// TIA Portal V20 export
TYPE "LKinCtrl_typeAdvPointers"
   STRUCT
      addPointer : DInt := 0;   // pointer to add new comds to PathData after cmd has been executed by MovePath
      retrievePointer : DInt := 0;   // pointer to show which cmd is the next to be retrieved by MovePath
      addPointerRestarted : Bool;   // addPointer restarted after overflow
      ignoreAddPointer : Bool := TRUE;   // addPointer not taken into account for buffering, unless set by previous data source
      bufferLocked : Bool;   // buffer locked to wait for previous data source - read data locked
      preprocessingStop : Bool;   // parser reached a preprocessing stop
   END_STRUCT;
END_TYPE
